// TIA Portal V20 export
TYPE "LER_typeAlignThetaCalibrationCommands"
// stored: Access Published
   STRUCT
      stepStart : Bool;
      stepStop : Bool;
      errorAck : Bool;
      Apply : Bool;
      MovePos1 : Bool;
      MovePos2 : Bool;
      MovePos3 : Bool;
   END_STRUCT;
END_TYPE
